Staubli VAL3: killAllTask.pgx

program killAllTask()
begin
  taskKill("Page")
  wait(taskStatus("Page")==-1)
  taskKill("Mot")
  wait(taskStatus("Mot")==-1)
  taskKill("sgd")
  wait(taskStatus("sgd")==-1)
end
